# EPICS substitutions: BLDApp/Db/eOrbitsFcomSXR.substitutions
file eOrbitsFcom.substitutions
{
  pattern
  { BPM1, BPM2, BPM3, BPM4, BPM5, BPM6, BPM7, BPM8, BPM9, BPM10, BPM11, EC }
  { BPMS:LTUS:860:, BPMS:LTUH:880:, BPMS:UNDS:1690:, BPMS:UNDS:1990:, BPMS:UNDS:2190:, BPMS:UNDS:2490:, BPMS:UNDS:2590:, BPMS:UNDS:2690:, BPMS:UNDS:2790:, BPMS:UNDS:2890:, BPMS:UNDS:2990:, $(EC)}

}
